TYPE DUT_HMI_07_MANUALS :
STRUCT
	PS : ARRAY[0..CNC.NUM_MAX_MANUALS_07-1] OF BOOL;
	LS : ARRAY[0..CNC.NUM_MAX_MANUALS_07-1] OF BOOL;
END_STRUCT
END_TYPE

(* stored: Version 1.1.0.1, ProductVersion 3.1.4024.13
   DUT DUT_HMI_07_MANUALS: Id {38947564-5e12-4d48-9b1b-e26b1abf6cff} *)
